(* Logix 5000 project; controller BTS01 vendor 1 type 14 code 217 rev 32.14; software revision 32.04; part 15 of 15 *)
(* tags used below, declared in another part *)
   C02S01 : REAL[8];   // 5069-IF8
   CIP_1_ACTIVE_PROGRAM : CIP_PROGRAM;
   CIP_1_ACTIVE_PROGRAM_SPANISH : CIP_PROGRAM;
   CIP_1_PROGRAMS_SPANISH : CIP_PROGRAM[20];
   CIP_1_RECIPE_SELECTED_SPANISH_HMI : STRING;
   CIPNames_Spanish : STRING[20];
   DummyString : STRING[10];
   DummyString2 : STRING[20];
   DummyString3 : STRING[20];
   Flow_Detected : BOOL;
   P1001 : DTE_VFD;   // Dressing Tank Fill Pump
   Pulse_DINT : DINT;
   TK1100_PID : PID;   // Tank 1100 Level Control
   TK1200_PID : PID;   // Tank 1200 Level Control
   TransferNames_Spanish : STRING[20];
   TransferOk : BOOL;
   TransferSelection : DINT;
   UnloadNames_Spanish : STRING[20];
(* MainProgram, continued *)

ROUTINE R13_Flow_Meter   (* ladder *)
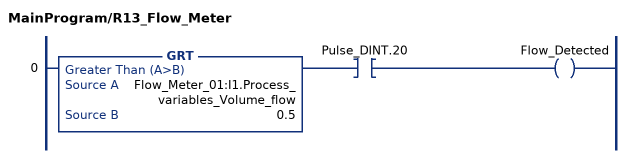
   0: GRT(Flow_Meter_01:I1.Process_variables_Volume_flow,0.5)XIC(Pulse_DINT.20)OTE(Flow_Detected);
END_ROUTINE

ROUTINE R20_P1001_PID   (* ladder *)
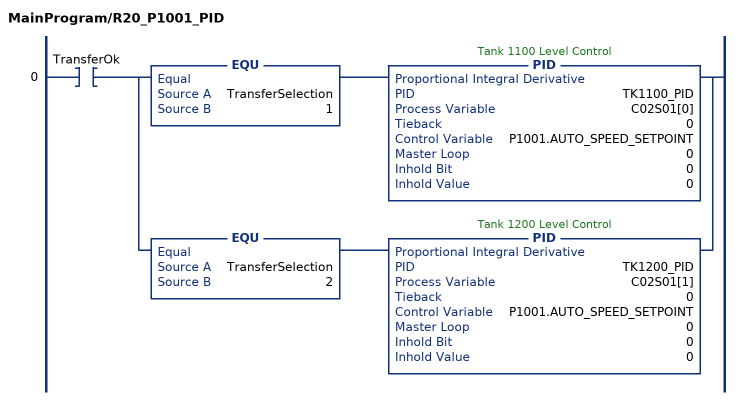
   0: XIC(TransferOk)[EQU(TransferSelection,1) PID(TK1100_PID,C02S01[0],0,P1001.AUTO_SPEED_SETPOINT,0,0,0) ,EQU(TransferSelection,2) PID(TK1200_PID,C02S01[1],0,P1001.AUTO_SPEED_SETPOINT,0,0,0) ];
END_ROUTINE

ROUTINE R30_TRANSLATION   (* ladder *)
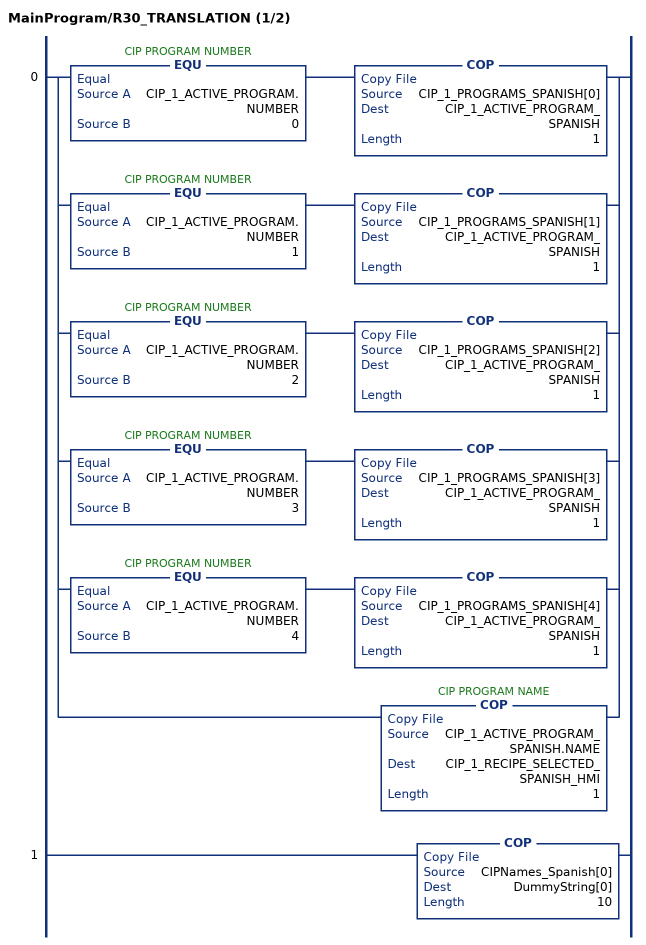
   0: [EQU(CIP_1_ACTIVE_PROGRAM.NUMBER,0) COP(CIP_1_PROGRAMS_SPANISH[0],CIP_1_ACTIVE_PROGRAM_SPANISH,1) ,EQU(CIP_1_ACTIVE_PROGRAM.NUMBER,1) COP(CIP_1_PROGRAMS_SPANISH[1],CIP_1_ACTIVE_PROGRAM_SPANISH,1) ,EQU(CIP_1_ACTIVE_PROGRAM.NUMBER,2) COP(CIP_1_PROGRAMS_SPANISH[2],CIP_1_ACTIVE_PROGRAM_SPANISH,1) ,EQU(CIP_1_ACTIVE_PROGRAM.NUMBER,3) COP(CIP_1_PROGRAMS_SPANISH[3],CIP_1_ACTIVE_PROGRAM_SPANISH,1) ,EQU(CIP_1_ACTIVE_PROGRAM.NUMBER,4) COP(CIP_1_PROGRAMS_SPANISH[4],CIP_1_ACTIVE_PROGRAM_SPANISH,1) ,COP(CIP_1_ACTIVE_PROGRAM_SPANISH.NAME,CIP_1_RECIPE_SELECTED_SPANISH_HMI,1) ];
   1: COP(CIPNames_Spanish[0],DummyString[0],10);
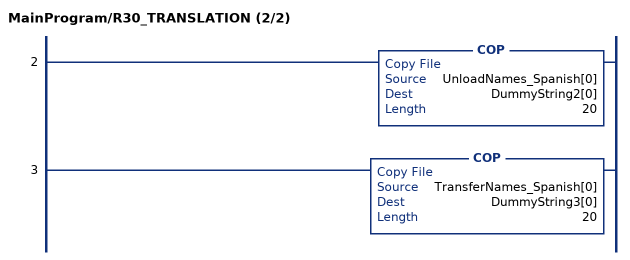
   2: COP(UnloadNames_Spanish[0],DummyString2[0],20);
   3: COP(TransferNames_Spanish[0],DummyString3[0],20);
END_ROUTINE
END_PROGRAM
